PROGRAM POUexecute
VAR
	iCount:INT;
	
	t1: TON;
	output: BOOL;
END_VAR

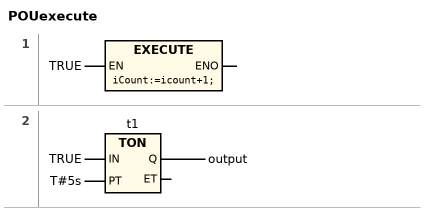
// NETWORK 1
iCount:=icount+1;

// NETWORK 2
t1(IN := TRUE, PT := T#5s); // TON
output := t1.Q;

END_PROGRAM

(* stored: Version 1.1.0.1, ProductVersion 3.1.4024.16
   POU POUexecute: Id {990f205a-b44a-4eb8-adf4-ef51ee7fa411}, SpecialFunc None *)
